FUNCTION_BLOCK EtherCatIoDevice EXTENDS CyclicComponent IMPLEMENTS I_EcIoDevice
VAR
	_Config		  : REFERENCE TO ST_EcSlaveConfigData;
	_State		  : REFERENCE TO ST_EcSlaveState;
	_SyncUnit	  : I_SyncUnitTask;
	_CoeScheduler : I_CoeTransferScheduler;
	_AmsAddr	  : AMSADDR;
	CoeDevice	  : CoeDevice('CoE Terminal');
	{attribute 'hide'}
	NullCoeDevice : NullCoeDevice('Null Terminal');
END_VAR

PROPERTY AmsNetId : AMSNETID
SET
_AmsAddr.netId := AmsNetId;
END_SET
END_PROPERTY

{attribute 'monitoring' := 'call'}
PROPERTY Bootstrap : BOOL
GET
VAR
	DiagByte : BYTE;
END_VAR
IF __ISVALIDREF(_State) THEN
	DiagByte  := _State.deviceState AND 16#0F;
	Bootstrap := DiagByte = EC_DEVICE_STATE_BOOTSTRAP;
END_IF
END_GET
END_PROPERTY

// CoE access of this slave; NullCoeDevice when the slave has no mailbox (or no configuration yet).
PROPERTY CoE : I_CoeDevice
GET
IF NOT __ISVALIDREF(_Config) OR_ELSE _Config.nMailboxInSize = 0 THEN
	CoE := NullCoeDevice;
ELSE
	CoE := CoeDevice;
END_IF
END_GET
SET
END_SET
END_PROPERTY

// Scheduler that services this slave's CoE transfers (set by EtherCatMaster during Initialize).
// Without one, CyclicLogic must be called each cycle while CoE.Busy.
PROPERTY CoeScheduler : I_CoeTransferScheduler
SET
_CoeScheduler		:= CoeScheduler;
CoeDevice.Scheduler := CoeScheduler;
END_SET
END_PROPERTY

PROPERTY Configuration : REFERENCE TO ST_EcSlaveConfigData
GET
Configuration REF= _Config;
END_GET
SET
_Config REF= Configuration;

(* The CoE mailbox is addressed by the EtherCAT address of the slave. *)
IF __ISVALIDREF(_Config) THEN
	_AmsAddr.port	  := _Config.nAddr;
	CoeDevice.AdsAddr REF= _AmsAddr;
END_IF
END_SET
END_PROPERTY

// Services a CoE transfer in flight when no CoeScheduler is attached. With a scheduler
// (the normal case under EtherCatMaster) this method does nothing.
METHOD CyclicLogic
IF _CoeScheduler <> 0 THEN
	RETURN;
END_IF

IF __ISVALIDREF(_Config) AND_THEN _Config.nMailboxInSize <> 0 AND_THEN CoeDevice.Busy THEN
	CoeDevice.CyclicLogic();
END_IF
END_METHOD

// EC_DEVICE_STATE_ERROR: state machine error in the slave (deviceState bit 4).
{attribute 'monitoring' := 'call'}
PROPERTY DeviceError : BOOL
GET
IF __ISVALIDREF(_State) THEN
	DeviceError := _State.deviceState.4;
END_IF
END_GET
END_PROPERTY

// EC_DEVICE_STATE_DISABLED: slave is disabled in the configuration (deviceState bit 7).
{attribute 'monitoring' := 'call'}
PROPERTY Disabled : BOOL
GET
IF __ISVALIDREF(_State) THEN
	Disabled := _State.deviceState.7;
END_IF
END_GET
END_PROPERTY

{attribute 'monitoring' := 'call'}
PROPERTY Init : BOOL
GET
VAR
	DiagByte : BYTE;
END_VAR
IF __ISVALIDREF(_State) THEN
	DiagByte := _State.deviceState AND 16#0F;
	Init	 := DiagByte = EC_DEVICE_STATE_INIT;
END_IF
END_GET
END_PROPERTY

// EC_DEVICE_STATE_INITCMD_ERROR: error while sending the init commands (deviceState bit 6).
{attribute 'monitoring' := 'call'}
PROPERTY InitCmdError : BOOL
GET
IF __ISVALIDREF(_State) THEN
	InitCmdError := _State.deviceState.6;
END_IF
END_GET
END_PROPERTY

// EC_DEVICE_STATE_INVALID_VPRS: vendor id / product code / revision / serial mismatch (deviceState bit 5).
{attribute 'monitoring' := 'call'}
PROPERTY InvalidVPRS : BOOL
GET
IF __ISVALIDREF(_State) THEN
	InvalidVPRS := _State.deviceState.5;
END_IF
END_GET
END_PROPERTY

{attribute 'monitoring' := 'call'}
PROPERTY IoDataValid : BOOL
GET
IF _SyncUnit <> 0 THEN
	IoDataValid := _SyncUnit.IoDataValid;
ELSE
	IoDataValid := TRUE;
END_IF
END_GET
END_PROPERTY

{attribute 'monitoring' := 'call'}
PROPERTY OP : BOOL
GET
VAR
	DiagByte : BYTE;
END_VAR
IF __ISVALIDREF(_State) THEN
	DiagByte := _State.deviceState AND 16#0F;
	OP		 := DiagByte = EC_DEVICE_STATE_OP;
END_IF
END_GET
END_PROPERTY

{attribute 'monitoring' := 'call'}
PROPERTY PreOp : BOOL
GET
VAR
	DiagByte : BYTE;
END_VAR
IF __ISVALIDREF(_State) THEN
	DiagByte := _State.deviceState AND 16#0F;
	PreOp	 := DiagByte = EC_DEVICE_STATE_PREOP;
END_IF
END_GET
END_PROPERTY

{attribute 'monitoring' := 'call'}
PROPERTY SafeOp : BOOL
GET
VAR
	DiagByte : BYTE;
END_VAR
IF __ISVALIDREF(_State) THEN
	DiagByte := _State.deviceState AND 16#0F;
	SafeOp	 := DiagByte = EC_DEVICE_STATE_SAFEOP;
END_IF
END_GET
END_PROPERTY

PROPERTY State : REFERENCE TO ST_EcSlaveState
GET
State REF= _State;
END_GET
SET
_State REF= State;
END_SET
END_PROPERTY

PROPERTY SyncUnit : I_SyncUnitTask
SET
_SyncUnit := SyncUnit;
END_SET
END_PROPERTY

END_FUNCTION_BLOCK

(* stored: Version 1.1.0.1, ProductVersion 3.1.4026.18
   POU EtherCatIoDevice: Id {20a9f0b1-40b0-400f-882c-783fc1cdd204}, SpecialFunc None
   Folder Device: Id {0e6012ac-dfb3-49bf-b9b6-e8b700a86eb0}
   Property AmsNetId: Id {59f5bcc5-b664-4721-8eaf-547a77cee820}
   Set Set: Id {d5ed1dac-2482-4982-aea9-09ea8fbe7c1c}
   Property Bootstrap: Id {6d8beaa5-7350-497a-9664-f92d86b4d56a}
   Get Get: Id {f78f2411-98e7-4c9f-af73-a9bef93883f8}
   Property CoE: Id {3571bd28-7a3f-4af9-8812-1e004a6a6323}
   Get Get: Id {4794d657-a8db-45a2-ae07-50370d61eb03}
   Set Set: Id {d80f7747-bb23-471e-b687-fad92a28aafe}
   Property CoeScheduler: Id {a22cba2b-bedc-4755-9198-5f47fc740806}
   Set Set: Id {d2a339a6-ef62-4492-bf33-dd64fbd4e5e9}
   Property Configuration: Id {5edeac0f-d414-4913-abd8-25629f2d8804}
   Get Get: Id {be8827bd-5394-49e0-8f69-08f4516e301e}
   Set Set: Id {bd8d5771-f645-4bf4-8e51-400374428bad}
   Method CyclicLogic: Id {4535afd1-41ad-4a0b-b50f-d26e99d4b7ce}
   Property DeviceError: Id {56a432d0-8bf0-4f61-9d42-0a3e7223eb04}
   Get Get: Id {8e068f78-253e-40c1-b647-f54cbf1caed7}
   Property Disabled: Id {ae3d4377-3250-4eac-9ae7-00e5e7d12533}
   Get Get: Id {c55405db-ab23-4a29-9f22-847edfd9b27f}
   Property Init: Id {22a145bc-7c97-405d-9076-bd3571e36ca0}
   Get Get: Id {b69da1bc-3e7f-4f52-bd17-ee243b3418e8}
   Property InitCmdError: Id {d8fd24df-4de2-4a2b-a273-c17c398db933}
   Get Get: Id {961f39f3-6722-49b2-a728-3587fcd7d26b}
   Property InvalidVPRS: Id {c5fd7491-68a3-46a1-aae0-d982fc628cd7}
   Get Get: Id {f76c247f-ff58-40dc-9782-54ac2c7b4c91}
   Property IoDataValid: Id {4a75f071-59af-4a48-9dc3-447db374b183}
   Get Get: Id {57d9357e-87be-49c0-aaf2-9d68b8f0a4bc}
   Property OP: Id {eb1f0a23-5ad4-40fc-871c-678fde62bc70}
   Get Get: Id {b16f5fba-237a-4c73-aae9-36674700194d}
   Property PreOp: Id {04485a59-96d0-4266-b1aa-a6d775b9b496}
   Get Get: Id {87665946-6a3f-4051-9cd0-9041a83b38d2}
   Property SafeOp: Id {61450f79-f493-43db-9d99-127882730b10}
   Get Get: Id {59907eae-6723-4af7-9151-005c94a3236f}
   Property State: Id {7a8d6550-1b78-406d-8ecd-7e25decdd9e3}
   Get Get: Id {cb6dd145-705e-42af-972f-1e157d39cc88}
   Set Set: Id {889dd6d0-b640-4d3f-8228-3e53c6b88c4c}
   Property SyncUnit: Id {cc8e8db4-5398-48e5-9950-6c3dff9c0ecd}
   Set Set: Id {09b0faa4-bd95-4576-b84c-17bcc77bbbc4} *)
